{attribute 'qualified_only'}
VAR_GLOBAL
	bOutput1 AT%Q* : BOOL;
END_VAR

(* stored: Version 1.1.0.1, ProductVersion 3.1.4024.12
   GVL GVL: Id {3f10fd27-8586-4e82-a4f9-14de1d30ab05} *)
